FUNCTION_BLOCK FB_HeatingNetworkHighTemperature
VAR_INPUT
	//control struct for hnht
	controlAutomatic : ST_HeatingNetworkHighTemperatureControl;	
	
	stAmbientState : ST_AmbientState;
END_VAR
VAR_OUTPUT
	{attribute 'OPC.UA.DA' := '1'}
	localState : ST_BufferStorageState;
END_VAR
VAR
	//systems
	BufferStorage : FB_BufferStorage;
	CHP1System : FB_CHPSystem;
	CHP2System : FB_CHPSystem;
	CondensingBoilerSystem : FB_CondensingBoilerSystem;
	StaticHeatingSystem : FB_StaticHeatingSystem;
	CentralMachineHeatingSystem : FB_HNHT_CentralMachineHeating;
	AnnealingOvenExhaustGasSystem : FB_AnnealingOvenExhaustGasSystem;
	
	stSV_SupplyAirDefaultParameters : ST_DiscreteValveDefaultParameters := (nFeedback := 0);
	SV_SupplyAir : FB_DiscreteValve := (ST_DefaultParameters := stSV_SupplyAirDefaultParameters);
		
	//machines
	MAFAC_Java : FB_MAFAC_Java;
	AnnealingOvenExhaustGas : FB_AnnealingOven;
	
	//internal variables
	bSetStatusOn_CentralMachineHeating : BOOL;
	bSetStatusOn_AnnealingOven : BOOL;
END_VAR

//buffer storage system
BufferStorage();
localState := BufferStorage.localState;

//producer
CHP1System(bSetStatusOnAutomatic := controlAutomatic.bSetStatusOn_CHP1,
	bAlgorithmPermission := controlAutomatic.bAlgorithmPermission,
	fSetPointAutomatic := controlAutomatic.fFeedTemperature,
	aHeatCounterTelegramm := Telegramm_WZ_BHKW_1,
	sIPAddressCHP := Global_IP_Adresses.BHKW_921_ModbusTCP);

CHP2System(bSetStatusOnAutomatic := controlAutomatic.bSetStatusOn_CHP2,
	bAlgorithmPermission := controlAutomatic.bAlgorithmPermission,
	fSetPointAutomatic := controlAutomatic.fFeedTemperature,
	aHeatCounterTelegramm := Telegramm_WZ_BHKW_2,
	sIPAddressCHP := Global_IP_Adresses.BHKW_922_ModbusTCP);

SV_SupplyAir.GetState_BI();
SV_SupplyAir(bSetStatusOnAutomatic := CHP1System.bSetStatusOnFeedback OR CHP2System.bSetStatusOnFeedback,
	bAlgorithmPermission := controlAutomatic.bAlgorithmPermission);
SV_SupplyAir.SetState_BO();

CondensingBoilerSystem(bSetStatusOnAutomatic := controlAutomatic.bSetStatusOn_CondensingBoiler,
	bAlgorithmPermission := controlAutomatic.bAlgorithmPermission,
	fSetPointAutomatic := controlAutomatic.fFeedTemperature);
				
//consumer
StaticHeatingSystem(bSetStatusOnAutomatic := controlAutomatic.bSetStatusOn_StaticHeating,
	bAlgorithmPermission := controlAutomatic.bAlgorithmPermission,
	fSetPointAutomatic := 0,
	stAmbientState := stAmbientState);
	
MAFAC_Java();
bSetStatusOn_CentralMachineHeating := MAFAC_Java.bStatusOn;
CentralMachineHeatingSystem(bSetStatusOnAutomatic := bSetStatusOn_CentralMachineHeating,
	bAlgorithmPermission := controlAutomatic.bAlgorithmPermission,
	fSetPointAutomatic := 80);
	
AnnealingOvenExhaustGas();
bSetStatusOn_AnnealingOven := AnnealingOvenExhaustGas.bStatusOn_ExhaustGas;
AnnealingOvenExhaustGasSystem(bSetStatusOnAutomatic := bSetStatusOn_AnnealingOven,
	bAlgorithmPermission := controlAutomatic.bAlgorithmPermission,
	fSetPointAutomatic := controlAutomatic.fFeedTemperature);

END_FUNCTION_BLOCK

(* stored: Version 1.1.0.1, ProductVersion 3.1.4024.10
   POU FB_HeatingNetworkHighTemperature: Id {2ced51e0-a3cc-4f43-8e53-7f6a9427e782}, SpecialFunc None *)
